TYPE ST_XtsMotorEtherCatDiag :
STRUCT
	fbSource : FB_TcSourceInfo;
	fbAlarmNotInOpMode : FB_TcAlarm;
	fbAlarmNoCommunication : FB_TcAlarm;
	
	fbGetSlaveState : FB_EcGetSlaveState;
	nLastState : BYTE;
END_STRUCT
END_TYPE

(* stored: Version 1.1.0.1, ProductVersion 3.1.4024.12
   DUT ST_XtsMotorEtherCatDiag: Id {a7f0d811-fc9b-427f-8b3d-13cbfaad5328} *)
